// SIMATIC S7-200 project (STEP 7-Micro/WIN), CPU 222 REL 02.01

SYMBOL_TABLE USER1
RUN_AUT0         M0.2     // SISTEMA IN RUN AUTOMATICO
SOSTA_SX         M0.1     // SOSTA PER SVUOTAMENTO
SOSTA_DX         M0.0     // SOSTA PER ILTEMPO DI RIEMPIMENTO
START            I0.0     // PULSANTE AVVIO CICLO
FC_SX            I0.1     // FINECORSA SINISTRO
CELL_SX          I0.2     // CONSENSO AL CARICO SULLA POSTAZIONE SINISTRA
FC_DX            I0.3     // FINECORSA DESTRO
CELL_DX          I0.4     // CONSENSO AL CARICO SULLA POSTAZIONE DESTRA
STOP_            I0.5     // PULSANTE DI ARESTO CICLO STOP
AUTO             I0.6     // ESECUZIONE DEL PROCESSO IN CICLO AUTOMATICO
MANU             I0.7     // ESECUZIONE DEL PROCESSO IN CICLO PASSO-PASSO
MOT_DX           Q0.0     // COMANDO MARCIA MOTORE VERSO DESTRA
MOT_SX           Q0.1     // COMANDO MARCIA MOTORE VERSO SINISTRA
EV_RIEMP         Q0.2     // COMANDO VALVOLA DI RIEMIMENTO
EV_SVUOT         Q0.3     // DISPOSITIVO IDRAULICO DI SVUOTAMENTO
END_SYMBOL_TABLE

ORGANIZATION_BLOCK MAIN:OB1
TITLE=DPS 205 TRASPORTO MATERIALE SFUSO
// 
BEGIN
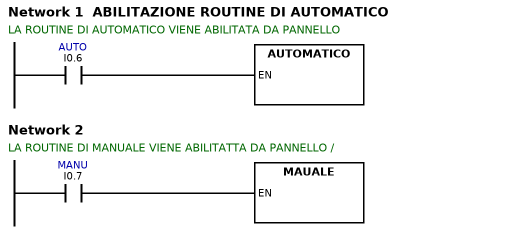
Network 1 // ABILITAZIONE ROUTINE DI AUTOMATICO
// LA ROUTINE DI AUTOMATICO VIENE ABILITATA DA PANNELLO
LD     AUTO:I0.6
CALL   AUTOMATICO:SBR0
Network 2
// LA ROUTINE DI MANUALE VIENE ABILITATTA DA PANNELLO
// 
LD     MANU:I0.7
CALL   MAUALE:SBR1
END_ORGANIZATION_BLOCK

SUBROUTINE_BLOCK AUTOMATICO:SBR0
TITLE=SUB ROUTINE AUTOMATICO
BEGIN
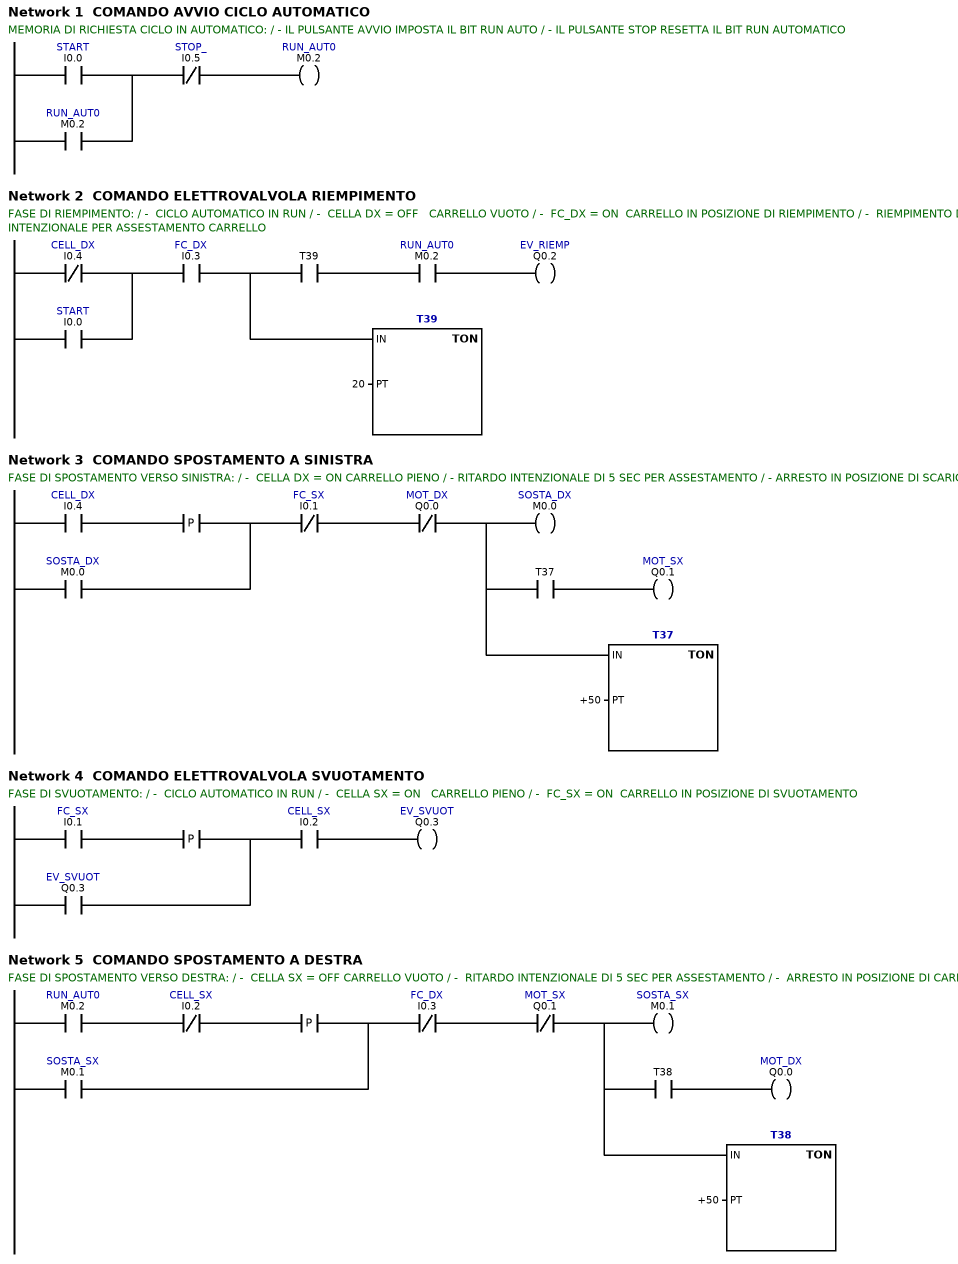
Network 1 // COMANDO AVVIO CICLO AUTOMATICO
// MEMORIA DI RICHIESTA CICLO IN AUTOMATICO:
// - IL PULSANTE AVVIO IMPOSTA IL BIT RUN AUTO
// - IL PULSANTE STOP RESETTA IL BIT RUN AUTOMATICO
LD     START:I0.0
O      RUN_AUT0:M0.2
AN     STOP_:I0.5
=      RUN_AUT0:M0.2
Network 2 // COMANDO ELETTROVALVOLA RIEMPIMENTO
// FASE DI RIEMPIMENTO:
// -  CICLO AUTOMATICO IN RUN
// -  CELLA DX = OFF   CARRELLO VUOTO
// -  FC_DX = ON  CARRELLO IN POSIZIONE DI RIEMPIMENTO
// -  RIEMPIMENTO DOPO RITARDO INTENZIONALE PER ASSESTAMENTO CARRELLO
LDN    CELL_DX:I0.4
O      START:I0.0
A      FC_DX:I0.3
LPS
A      T39
A      RUN_AUT0:M0.2
=      EV_RIEMP:Q0.2
LPP
TON    T39, 20
Network 3 // COMANDO SPOSTAMENTO A SINISTRA
// FASE DI SPOSTAMENTO VERSO SINISTRA:
// -  CELLA DX = ON CARRELLO PIENO
// - RITARDO INTENZIONALE DI 5 SEC PER ASSESTAMENTO
// - ARRESTO IN POSIZIONE DI SCARICO FC_SX = ON
LD     CELL_DX:I0.4
EU     0
O      SOSTA_DX:M0.0
AN     FC_SX:I0.1
AN     MOT_DX:Q0.0
LPS
=      SOSTA_DX:M0.0
A      T37
=      MOT_SX:Q0.1
LPP
TON    T37, +50
Network 4 // COMANDO ELETTROVALVOLA SVUOTAMENTO
// FASE DI SVUOTAMENTO:
// -  CICLO AUTOMATICO IN RUN
// -  CELLA SX = ON   CARRELLO PIENO
// -  FC_SX = ON  CARRELLO IN POSIZIONE DI SVUOTAMENTO
LD     FC_SX:I0.1
EU     1
O      EV_SVUOT:Q0.3
A      CELL_SX:I0.2
=      EV_SVUOT:Q0.3
Network 5 // COMANDO SPOSTAMENTO A DESTRA
// FASE DI SPOSTAMENTO VERSO DESTRA:
// -  CELLA SX = OFF CARRELLO VUOTO
// -  RITARDO INTENZIONALE DI 5 SEC PER ASSESTAMENTO
// -  ARRESTO IN POSIZIONE DI CARICO FC_DX = ON
LD     RUN_AUT0:M0.2
AN     CELL_SX:I0.2
EU     2
O      SOSTA_SX:M0.1
AN     FC_DX:I0.3
AN     MOT_SX:Q0.1
LPS
=      SOSTA_SX:M0.1
A      T38
=      MOT_DX:Q0.0
LPP
TON    T38, +50
END_SUBROUTINE_BLOCK

SUBROUTINE_BLOCK MAUALE:SBR1
TITLE=COMMENTI SUL SOTTOPROGRAMMA
BEGIN
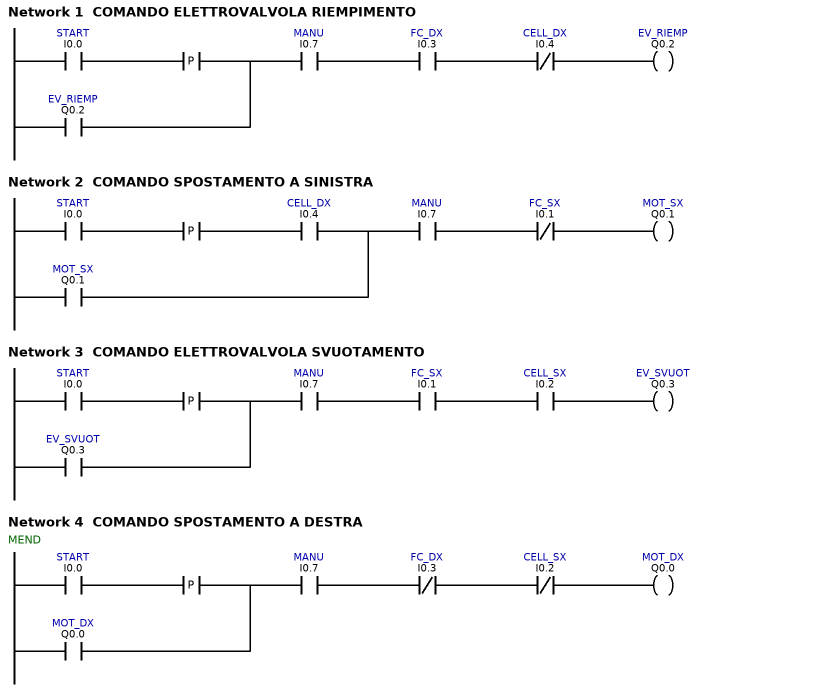
Network 1 // COMANDO ELETTROVALVOLA RIEMPIMENTO
LD     START:I0.0
EU     3
O      EV_RIEMP:Q0.2
A      MANU:I0.7
A      FC_DX:I0.3
AN     CELL_DX:I0.4
=      EV_RIEMP:Q0.2
Network 2 // COMANDO SPOSTAMENTO A SINISTRA
LD     START:I0.0
EU     4
A      CELL_DX:I0.4
O      MOT_SX:Q0.1
A      MANU:I0.7
AN     FC_SX:I0.1
=      MOT_SX:Q0.1
Network 3 // COMANDO ELETTROVALVOLA SVUOTAMENTO
LD     START:I0.0
EU     5
O      EV_SVUOT:Q0.3
A      MANU:I0.7
A      FC_SX:I0.1
A      CELL_SX:I0.2
=      EV_SVUOT:Q0.3
Network 4 // COMANDO SPOSTAMENTO A DESTRA
// MEND
LD     START:I0.0
EU     6
O      MOT_DX:Q0.0
A      MANU:I0.7
AN     FC_DX:I0.3
AN     CELL_SX:I0.2
=      MOT_DX:Q0.0
Network 5 // Ti
// Commento del segmento
END_SUBROUTINE_BLOCK
